TYPE ST_RGBW_Zustand :
STRUCT
	Betrieb	: BOOL;
	R_Wert	: REAL;
	G_Wert	: REAL;
	B_Wert	: REAL;
	W_Wert	: REAL;
END_STRUCT
END_TYPE

(* stored: Version 1.1.0.1, ProductVersion 3.1.4024.9
   DUT ST_RGBW_Zustand: Id {ca9dc1e1-1fb1-4373-a56d-d94498421270} *)
